% RSLogix 500 project INTRO TO PLC - JOB 19.RSS, saved by version 10.00.00.00 %
PROJECT "PL06B"    % processor: Bul.1763 MicroLogix 1100 Series B %

PROGRAM FILES
  LAD 2   9 rungs

DATA FILES
  O0 OUTPUT  4 elements
  I1 INPUT  6 elements
  S2 STATUS  66 elements
  B3 BINARY  1 elements
  T4 TIMER  10 elements
  C5 COUNTER  2 elements
  R6 CONTROL  1 elements
  N7 INTEGER  5 elements
  F8 FLOAT  1 elements

LADDER 2
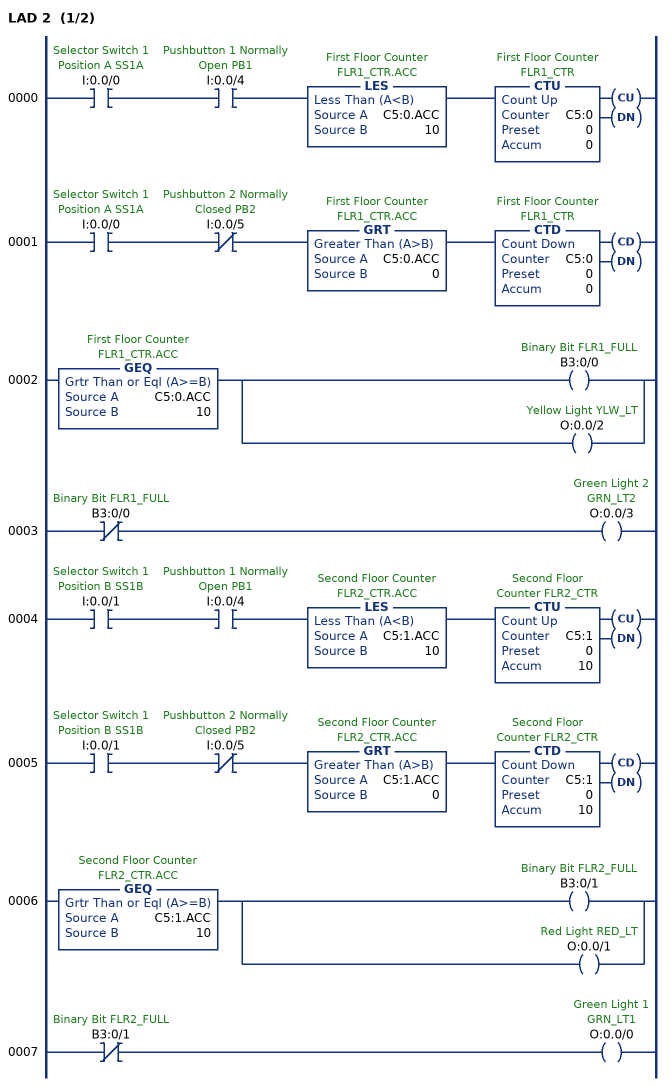
% Rung: 0 %
SOR XIC I:0.0/0 XIC I:0.0/4 LES C5:0.ACC 10 CTU C5:0 0 0 EOR
%   I:0.0/0  SS1A  "Selector Switch 1 Position A" %
%   I:0.0/4  PB1  "Pushbutton 1 Normally Open" %
%   C5:0  FLR1_CTR  "First Floor Counter" %
% Rung: 1 %
SOR XIC I:0.0/0 XIO I:0.0/5 GRT C5:0.ACC 0 CTD C5:0 0 0 EOR
%   I:0.0/0  SS1A  "Selector Switch 1 Position A" %
%   I:0.0/5  PB2  "Pushbutton 2 Normally Closed" %
%   C5:0  FLR1_CTR  "First Floor Counter" %
% Rung: 2 %
SOR GEQ C5:0.ACC 10 BST OTE B3:0/0 NXB OTE O:0.0/2 BND EOR
%   C5:0  FLR1_CTR  "First Floor Counter" %
%   B3:0/0  FLR1_FULL  "Binary Bit" %
%   O:0.0/2  YLW_LT  "Yellow Light" %
% Rung: 3 %
SOR XIO B3:0/0 OTE O:0.0/3 EOR
%   B3:0/0  FLR1_FULL  "Binary Bit" %
%   O:0.0/3  GRN_LT2  "Green Light 2" %
% Rung: 4 %
SOR XIC I:0.0/1 XIC I:0.0/4 LES C5:1.ACC 10 CTU C5:1 0 10 EOR
%   I:0.0/1  SS1B  "Selector Switch 1 Position B" %
%   I:0.0/4  PB1  "Pushbutton 1 Normally Open" %
%   C5:1  FLR2_CTR  "Second Floor Counter" %
% Rung: 5 %
SOR XIC I:0.0/1 XIO I:0.0/5 GRT C5:1.ACC 0 CTD C5:1 0 10 EOR
%   I:0.0/1  SS1B  "Selector Switch 1 Position B" %
%   I:0.0/5  PB2  "Pushbutton 2 Normally Closed" %
%   C5:1  FLR2_CTR  "Second Floor Counter" %
% Rung: 6 %
SOR GEQ C5:1.ACC 10 BST OTE B3:0/1 NXB OTE O:0.0/1 BND EOR
%   C5:1  FLR2_CTR  "Second Floor Counter" %
%   B3:0/1  FLR2_FULL  "Binary Bit" %
%   O:0.0/1  RED_LT  "Red Light" %
% Rung: 7 %
SOR XIO B3:0/1 OTE O:0.0/0 EOR
%   B3:0/1  FLR2_FULL  "Binary Bit" %
%   O:0.0/0  GRN_LT1  "Green Light 1" %

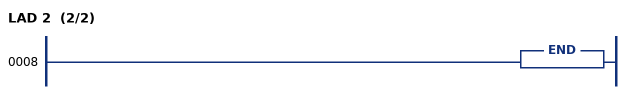
% Rung: 8 %
SOR END EOR

OTHER DOCUMENTED ADDRESSES
  B3:0/2  YLW_STOP  "Yellow Light Stop"
  B3:0/3  RED_STOP  "Red Light Stop"
  B3:0/4  GRN_STOP  "Green Light 1 Stop"
  B3:0/15  SCRATCH  "Scratch Bit"
  B3:1/1  RED_TMR_DNS  "Red Light Timer Done Storage"
  I  
  I:0.0/2  SS2A  "Selector Switch 2 Position A"
  I:0.0/3  SS2B  "Selector Switch 2 Position B"
  RTC:0.YR  RTC
  SEL1B  
  T4:0  INT_TMR  "Light Timer"
  T4:1  YLW_TMR  "Yellow Light Timer"
  T4:2  GRN_TMR  "Green Light Timer"
  T4:3  RST_TMR  "Reset Timer"

COMMENTS NOT ATTACHED TO A CURRENT RUNG
  B3:0/0: Typical Stop Start Logic

DATA TABLE (non-zero values as saved)
DATA B3
% B3:0 % 0X800A
DATA T4
% .PRE .ACC %
% T4:0 % 40 0
% T4:1 % 5 0
% T4:2 % 5 0
% T4:3 % 10 0
DATA C5
% .PRE .ACC %
% C5:1 % 0 10
DATA N7
% N7:0 % 555 0 0 0 0
